{attribute 'qualified_only'}
{attribute 'strict'}
{attribute 'to_string'}
TYPE ENUM_Fahrsystem :
(
	Warten := 0,
	Sicherheitscheck := 1,
	ZumStartStockwerk := 2,
	Tueren := 3,
	ZumZielStockwerk := 4,
	Aufstartablauf := 5
);
END_TYPE

(* stored: Version 1.1.0.1
   DUT ENUM_Fahrsystem: Id {1fcefb87-6428-4f2d-9511-e07c57150bbc} *)
